// TIA Portal V17 export
// export: Created 2023-12-22T15:02:58.9861649Z, ExportSetting WithDefaults, DisplayName Totally Integrated Automation Portal, DisplayVersion V17, DisplayName TIA Portal Openness, DisplayVersion V17, DisplayName TIA Portal Version Control Interface, DisplayVersion V17, DisplayName STEP 7 Professional, DisplayVersion V17, DisplayName STEP 7 Safety, DisplayVersion V17, DisplayName WinCC Advanced, DisplayVersion V17
FUNCTION_BLOCK "Main_Logick"   // FB1, LAD
{ S7_Optimized_Access := 'FALSE' }
VERSION : 0.1
// stored: AutoNumber true, IsIECCheckEnabled false, SetENOAutomatically false, UDAEnableTagReadback false
   VAR
      Time_Contrast_SKV { S7_SetPoint := 'True'} : "Time_D";   // Время сравнения наработки скважин (3 дня)
   END_VAR
   // Time_Contrast_SKV.SP_D := 3;
BEGIN

REGION Network 5
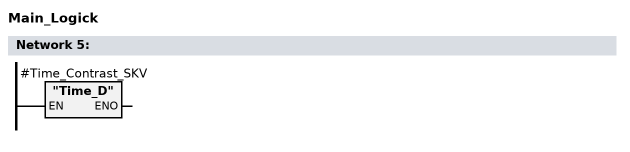
   RUNG wire#powerrail
      #Time_Contrast_SKV()
   END_RUNG
   // the same network as SCL:
   #Time_Contrast_SKV();   // "Time_D"
END_REGION
END_FUNCTION_BLOCK
